FUNCTION_BLOCK FB_EL922x_ChannelExtended IMPLEMENTS ITF_EL922x_ChannelExtended
VAR_INPUT
END_VAR
VAR_OUTPUT
END_VAR
VAR
	_Chn : EL922x_ChannelExtended;
END_VAR


PROPERTY DisabledByDI : BOOL
GET
DisabledByDI := _Chn.Status.DisabledByDI;
END_GET
END_PROPERTY


PROPERTY DisabledByOutput : BOOL
GET
DisabledByOutput := _Chn.Status.DisabledByOutput;
END_GET
END_PROPERTY


PROPERTY DisabledBySwitch : BOOL
GET
DisabledBySwitch := _Chn.Status.DisabledBySwitch;
END_GET
END_PROPERTY


PROPERTY Overload : BOOL
GET
Overload := _Chn.Status.Overload;
END_GET
END_PROPERTY


PROPERTY Overvoltage : BOOL
GET
Overvoltage := _Chn.Status.Overvoltage;
END_GET
END_PROPERTY


PROPERTY ShortCircuit : BOOL
GET
ShortCircuit := _Chn.Status.ShortCircuit;
END_GET
END_PROPERTY


PROPERTY StateDeviceSwitch : BOOL
GET
StateDeviceSwitch := _Chn.Status.StateDeviceSwitch;
END_GET
END_PROPERTY


PROPERTY StateDigitalInput : BOOL
GET
StateDigitalInput := _Chn.Status.StateDigitalInput;
END_GET
END_PROPERTY


PROPERTY Undervoltage : BOOL
GET
Undervoltage := _Chn.Status.Undervoltage;
END_GET
END_PROPERTY

END_FUNCTION_BLOCK

(* stored: Version 1.1.0.1, ProductVersion 3.1.4024.5
   POU FB_EL922x_ChannelExtended: Id {9757487c-991c-4df2-9a74-8898cc78a011}, SpecialFunc None
   Property DisabledByDI: Id {2150f53c-023b-4828-bdb2-98cb9d13e37e}
   Get Get: Id {d51d9500-f825-47d9-819d-b13e41232920}
   Property DisabledByOutput: Id {49f0e1d6-d31a-4a95-a0b1-f022ee3c0537}
   Get Get: Id {beed161c-dbe7-4ef4-8576-41104c020510}
   Property DisabledBySwitch: Id {1a824d32-5cc9-491e-a5e2-e068b8d7adc3}
   Get Get: Id {d0922947-56fe-4875-a8b3-28f631092c80}
   Property Overload: Id {347322a6-d7e5-4ecc-bd2c-eae47d597746}
   Get Get: Id {0c479487-50e2-41b4-b043-ded7d4bd097a}
   Property Overvoltage: Id {e4a6bc9a-5932-44c2-bb0f-76e22b4abdd1}
   Get Get: Id {8647ee9c-f952-46d5-8d97-330b212329ab}
   Property ShortCircuit: Id {c0944107-7473-421b-ba5d-e276cd557859}
   Get Get: Id {12dc32a6-c5aa-40a4-ae7b-8481020716f7}
   Property StateDeviceSwitch: Id {23d5908e-a535-40bd-8f0c-98f229a4c522}
   Get Get: Id {3869f6c2-6d66-49ba-8989-52ed95fabc69}
   Property StateDigitalInput: Id {0b18c46a-920b-4768-949a-361670587027}
   Get Get: Id {e37f2dd0-1b77-4e7e-a2bf-b0ad36f83bdc}
   Property Undervoltage: Id {c3be64b5-cefc-47cb-8b99-abcf7e0db533}
   Get Get: Id {efbc00d4-c70c-4d5e-9575-7511dec31a39} *)
